//{attribute 'qualified_only'}
//{attribute 'strict'}
TYPE E_User :
(
	eUser_none := 0,	(*User | none*)
	eUser_1,			(*User | 1*)
	eUser_2,			(*User | 2*)
	eUser_3,			(*User | 3*)
	eUser_4,			(*User | 4*)
	eUser_5,			(*User | 5*)
	eUser_6,			(*User | 6*)
	eUser_7,			(*User | 7*)
	eUser_8,			(*User | 8*)
	eUser_9,			(*User | 9*)
	eUser_10,			(*User | 10*)

	eUser_11,			(*User | 11*)
	eUser_12,			(*User | 12*)
	eUser_13,			(*User | 13*)
	eUser_14,			(*User | 14*)
	eUser_15,			(*User | 15*)
	eUser_16,			(*User | 16*)
	eUser_17,			(*User | 17*)
	eUser_18,			(*User | 18*)
	eUser_19,			(*User | 19*)
	eUser_20,			(*User | 20*)	
(*Maximum*)
	eUser_nMaxIdx
);
END_TYPE

(* stored: Version 1.1.0.1
   EnumerationTextList E_User: Id {5ccde2d0-2ce4-4b7c-a417-4862af46f61d} *)
